//==================================================================================================
//							Beckhoff Automation Poland
//									10.01.2019
//	Wszystkomajacy blok funkcyjny do sterowania osia, 
//	wymagane biblioteki: Tc2_MC2, Tc2_Utilities
// 	v1.0 	|| TC v 3.1.4022.27	 	|| - first edition
//==================================================================================================
{attribute 'reflection'}
FUNCTION_BLOCK FB_McAxisOnlineNC
VAR_IN_OUT
	stMcAxisOnline						: ST_McAxisOnline;
	Axis								: AXIS_REF;
END_VAR
VAR
	mcPower								: MC_Power;
	mcStop								: MC_Stop;
	mcHalt								: MC_Halt;
	mcStopSS1							: MC_Stop;
	mcStopSS2							: MC_Stop;
	mcReset								: MC_Reset;
	mcHome								: MC_Home;
	mcSetPosition						: MC_SetPosition;
	mcJog								: MC_Jog;

	mcMoveAbsolute						: MC_MoveAbsolute;
	mcMoveRelative						: MC_MoveRelative;
	mcMoveVelocity						: MC_MoveVelocity;
	mcMoveModulo						: MC_MoveModulo;
	mcMoveAbsolute2						: MC_MoveAbsolute;
	mcMoveRelative2						: MC_MoveRelative;
	mcMoveVelocity2						: MC_MoveVelocity;
	mcMoveModulo2						: MC_MoveModulo;

	fbNcLimitSwitch						: FB_NcSWLimitSwitchCtrl;
	mcReadParameterSet					: MC_ReadParameterSet;
	// Internal
	bInitialized						: BOOL;
			
	// Initialization
	iInitStep							: INT;
	bInitializationError				: BOOL;
	wInitializationErrorCounter			: WORD;
	bReadParameterSetReady				: BOOL;
	tonDelay							: TON;
	// Re init
	udiOnlineChangeCntOld				: UDINT;
	bOnlineChangeDetected				: BOOL;
	bReInit								: BOOL;
	bReInitialized						: BOOL;
	bReInitializationError				: BOOL;
	{attribute 'instance-path'}
	{attribute 'noinit'}
	sInstancePath						: STRING;
END_VAR

// Device dependent initialization 
ACT_Initialization();
// Device independent commands, mostly NC 
ACT_States();
ACT_SWLimitSwitch();
ACT_Stop();
ACT_Power();
ACT_Homing();
ACT_Jog();
ACT_Move();
ACT_ResetAndDiag();
ACT_SetPosition();
// Device independent error collection
ACT_ErrorCollection();

ACTION ACT_ErrorCollection:
// Error flags
stMcAxisOnline.stError.bDriveError					:= Axis.Status.DriveDeviceError;

stMcAxisOnline.stError.bNcError						:= Axis.Status.Error;

stMcAxisOnline.stError.bFBError						:= stMcAxisOnline.mcPower.bError OR stMcAxisOnline.mcReset.bError OR stMcAxisOnline.mcHome.bError OR stMcAxisOnline.mcJog.bError
													OR stMcAxisOnline.mcHalt.bError OR stMcAxisOnline.mcStop.bError OR stMcAxisOnline.mcSS1.bError OR stMcAxisOnline.mcSS2.bError
													OR stMcAxisOnline.mcMoveAbsolute.bError OR stMcAxisOnline.mcMoveRelative.bError OR stMcAxisOnline.mcMoveVelocity.bError OR stMcAxisOnline.mcMoveModulo.bError
													OR stMcAxisOnline.mcMoveAbsolute2.bError OR stMcAxisOnline.mcMoveRelative2.bError OR stMcAxisOnline.mcMoveVelocity2.bError OR stMcAxisOnline.mcMoveModulo2.bError
													OR stMcAxisOnline.stNcLimitSwitch.bError OR stMcAxisOnline.mcSetPosition.bError;
									
stMcAxisOnline.stError.bCommunicationError			:= stMcAxisOnline.stChannelErrorCode.bError OR stMcAxisOnline.stSetPositionOffset.bError OR stMcAxisOnline.stMotorMonitoring.bError OR stMcAxisOnline.stHoldingBrake.bError;

stMcAxisOnline.stError.bError						:= stMcAxisOnline.stError.bDriveError OR stMcAxisOnline.stError.bNcError OR stMcAxisOnline.stError.bFBError OR stMcAxisOnline.stError.bCommunicationError;
stMcAxisOnline.bError								:= stMcAxisOnline.stError.bError; // Forward one stage up

// Error codes
stMcAxisOnline.stError.uiDriveErrorID 				:= stMcAxisOnline.stChannelErrorCode.uiChannelErrorCode;
stMcAxisOnline.stError.uiDriveErrorIDHex 			:= stMcAxisOnline.stChannelErrorCode.uiChannelErrorCodeHex;

stMcAxisOnline.stError.udiNcErrorID 				:= Axis.Status.ErrorID;
stMcAxisOnline.stError.udiNcErrorIDHex 				:= Axis.Status.ErrorID;
	

stMcAxisOnline.stError.udiFBErrorID 				:= 	stMcAxisOnline.mcPower.udiErrorID + 
														stMcAxisOnline.mcReset.udiErrorID + 
														stMcAxisOnline.mcHome.udiErrorID + 
														stMcAxisOnline.mcJog.udiErrorID +
														stMcAxisOnline.mcHalt.udiErrorID + 
														stMcAxisOnline.mcStop.udiErrorID + 
														stMcAxisOnline.mcSS1.udiErrorID + 
														stMcAxisOnline.mcSS2.udiErrorID +
														stMcAxisOnline.mcMoveAbsolute.udiErrorID + 
														stMcAxisOnline.mcMoveRelative.udiErrorID + 
														stMcAxisOnline.mcMoveVelocity.udiErrorID + 
														stMcAxisOnline.mcMoveModulo.udiErrorID +
														stMcAxisOnline.mcMoveAbsolute2.udiErrorID + 
														stMcAxisOnline.mcMoveRelative2.udiErrorID + 
														stMcAxisOnline.mcMoveVelocity2.udiErrorID + 
														stMcAxisOnline.mcMoveModulo2.udiErrorID +
														stMcAxisOnline.stNcLimitSwitch.udiErrorID + 
														stMcAxisOnline.mcSetPosition.udiErrorID;

stMcAxisOnline.stError.udiFBErrorIDHex 				:= stMcAxisOnline.stError.udiFBErrorID;

stMcAxisOnline.stError.udiErrorID					:= stMcAxisOnline.stSetPositionOffset.udiErrorID;
stMcAxisOnline.stError.uiAdsErrorID					:= stMcAxisOnline.stChannelErrorCode.uiAdsErrId + stMcAxisOnline.stMotorMonitoring.uiAdsErrId + stMcAxisOnline.stHoldingBrake.uiAdsErrId;
stMcAxisOnline.stError.uiSecErrorID					:= stMcAxisOnline.stChannelErrorCode.uiSecErrId + stMcAxisOnline.stMotorMonitoring.uiSecErrId + stMcAxisOnline.stHoldingBrake.uiSecErrId;

stMcAxisOnline.stError.sNcError						:= F_AxErrMsg(stMcAxisOnline.stError.udiNcErrorID);
stMcAxisOnline.stError.sDriveError					:= F_AX5xErrMsg(stMcAxisOnline.stError.uiDriveErrorID);
END_ACTION

ACTION ACT_Homing:
mcHome(		Axis						:= Axis,
			Execute						:= stMcAxisOnline.mcHome.bExecute,
			Position					:= stMcAxisOnline.mcHome.lrPosition,
			HomingMode					:= stMcAxisOnline.mcHome.eHomingMode,
			BufferMode					:= stMcAxisOnline.mcHome.eBufferMode,
			Options						:= stMcAxisOnline.mcHome.stOptions,
			bCalibrationCam				:= stMcAxisOnline.mcHome.bCalibrationCam,
			Done						=> stMcAxisOnline.mcHome.bDone,
			Busy						=> stMcAxisOnline.mcHome.bBusy,
			Active						=> stMcAxisOnline.mcHome.bActive,
			CommandAborted				=> stMcAxisOnline.mcHome.bCommandAborted,
			Error						=> stMcAxisOnline.mcHome.bError,
			ErrorID						=> stMcAxisOnline.mcHome.udiErrorID);
END_ACTION

ACTION ACT_Initialization:
// bInitialized flag is set just once. 
// bReInitialized ise set each time we do online change or request reinit operation
// bDriveAddressReady, bReadParameterSetReady, bDriveRefReady - set just once after successed read

// Online change detection
bOnlineChangeDetected					:= udiOnlineChangeCntOld <> _AppInfo.OnlineChangeCnt;
udiOnlineChangeCntOld 					:= _AppInfo.OnlineChangeCnt;
// Reset init
IF bReInit OR bOnlineChangeDetected THEN
	iInitStep							:= 0;
END_IF

//Initialization process
CASE iInitStep OF
	0:	// Read Parameter Set
		
		stMcAxisOnline.mcReadParameterSet.bExecute		:=	 TRUE;
		iInitStep						:= iInitStep + 10;
		
	10: // Wait for data
	
		IF NOT stMcAxisOnline.mcReadParameterSet.bBusy THEN
			stMcAxisOnline.mcReadParameterSet.bExecute	:=	 FALSE;
			IF stMcAxisOnline.mcReadParameterSet.bDone THEN
				iInitStep 				:= iInitStep + 10;
				bReadParameterSetReady 	:= TRUE;
			ELSE
				iInitStep 				:= 1000;		// Error step
			END_IF
		END_IF	
	
	20: // Success - initialized flag, clear error
		bReInitialized					:= bInitialized;	// TRUE only when it's not first initialization e.g. online change
		bInitialized 					:= TRUE;
		bReInitializationError			:= FALSE;			// TRUE only when it's not first initialization e.g. online change
		bInitializationError			:= FALSE;
		iInitStep 						:= iInitStep + 10;
		
	30: // Idle
	
		;
		
	1000: // Error step
		wInitializationErrorCounter 	:= wInitializationErrorCounter + 1;
		IF wInitializationErrorCounter < 100 THEN
			iInitStep					:= iInitStep + 5;			// Go to delay
		ELSE
			bReInitializationError		:= bInitializationError;	// TRUE only when it's not first initialization e.g. online change
			bInitializationError		:= TRUE;
			bReInitialized				:= FALSE;
			iInitStep 					:= iInitStep + 10;
		END_IF

	1005: // Delay step
		tonDelay(IN:= TRUE, PT:= T#1S);
		IF tonDelay.Q THEN
			tonDelay(IN:= FALSE, PT:= T#1S);
			iInitStep					:= 0;
		END_IF
		
	1010: // Idle after error
		;
	
END_CASE
				
mcReadParameterSet(	Parameter			:= stMcAxisOnline.stAxisParameter,
					Axis				:= Axis,
					Execute				:= stMcAxisOnline.mcReadParameterSet.bExecute,
					Done				=> stMcAxisOnline.mcReadParameterSet.bDone,
					Busy				=> stMcAxisOnline.mcReadParameterSet.bBusy,
					Error				=> stMcAxisOnline.mcReadParameterSet.bError,
					ErrorID				=> stMcAxisOnline.mcReadParameterSet.udiErrorID);
END_ACTION

ACTION ACT_Jog:
// Direct access from bSlow or bFast, if none then free choice
IF stMcAxisOnline.mcJog.bSlowForward OR stMcAxisOnline.mcJog.bSlowBackward THEN
	stMcAxisOnline.mcJog.eMode			:= MC_JOGMODE_STANDARD_SLOW;
ELSIF stMcAxisOnline.mcJog.bFastForward OR stMcAxisOnline.mcJog.bFastBackward THEN
	stMcAxisOnline.mcJog.eMode			:= MC_JOGMODE_STANDARD_FAST;
END_IF

mcJog(		Axis						:= Axis,
			JogForward					:= stMcAxisOnline.mcJog.bJogForward OR stMcAxisOnline.mcJog.bSlowForward OR stMcAxisOnline.mcJog.bFastForward,
			JogBackwards				:= stMcAxisOnline.mcJog.bJogBackwards OR stMcAxisOnline.mcJog.bSlowBackward OR stMcAxisOnline.mcJog.bFastBackward,
			Mode						:= stMcAxisOnline.mcJog.eMode,
			Position					:= stMcAxisOnline.mcJog.lrPosition,
			Velocity					:= stMcAxisOnline.mcJog.lrVelocity,
			Acceleration				:= stMcAxisOnline.mcJog.lrAcceleration,
			Deceleration				:= stMcAxisOnline.mcJog.lrDeceleration,
			Jerk						:= stMcAxisOnline.mcJog.lrJerk,
			Done						=> stMcAxisOnline.mcJog.bDone,
			Busy						=> stMcAxisOnline.mcJog.bBusy,
			Active						=> stMcAxisOnline.mcJog.bActive,
			CommandAborted				=> stMcAxisOnline.mcJog.bCommandAborted,
			Error						=> stMcAxisOnline.mcJog.bError,
			ErrorID						=> stMcAxisOnline.mcJog.udiErrorID);
END_ACTION

ACTION ACT_Move:
{region "Primary"}
mcMoveAbsolute(	Axis					:= Axis,
				Execute					:= stMcAxisOnline.mcMoveAbsolute.bExecute,
				Position				:= stMcAxisOnline.mcMoveAbsolute.lrPosition,
				Velocity				:= stMcAxisOnline.mcMoveAbsolute.lrVelocity,
				Acceleration			:= stMcAxisOnline.mcMoveAbsolute.lrAcceleration,
				Deceleration			:= stMcAxisOnline.mcMoveAbsolute.lrDeceleration,
				Jerk					:= stMcAxisOnline.mcMoveAbsolute.lrJerk,
				BufferMode				:= stMcAxisOnline.mcMoveAbsolute.eBufferMode,
				Options					:= stMcAxisOnline.mcMoveAbsolute.stOptions,
				Done					=> stMcAxisOnline.mcMoveAbsolute.bDone,
				Busy					=> stMcAxisOnline.mcMoveAbsolute.bBusy,
				Active					=> stMcAxisOnline.mcMoveAbsolute.bActive,
				CommandAborted			=> stMcAxisOnline.mcMoveAbsolute.bCommandAborted,
				Error					=> stMcAxisOnline.mcMoveAbsolute.bError,
				ErrorID					=> stMcAxisOnline.mcMoveAbsolute.udiErrorID);

mcMoveRelative(	Axis					:= Axis,
				Execute					:= stMcAxisOnline.mcMoveRelative.bExecute,
				Distance				:= stMcAxisOnline.mcMoveRelative.lrDistance,
				Velocity				:= stMcAxisOnline.mcMoveRelative.lrVelocity,
				Acceleration			:= stMcAxisOnline.mcMoveRelative.lrAcceleration,
				Deceleration			:= stMcAxisOnline.mcMoveRelative.lrDeceleration,
				Jerk					:= stMcAxisOnline.mcMoveRelative.lrJerk,
				BufferMode				:= stMcAxisOnline.mcMoveRelative.eBufferMode,
				Options					:= stMcAxisOnline.mcMoveRelative.stOptions,
				Done					=> stMcAxisOnline.mcMoveRelative.bDone,
				Busy					=> stMcAxisOnline.mcMoveRelative.bBusy,
				Active					=> stMcAxisOnline.mcMoveRelative.bActive,
				CommandAborted			=> stMcAxisOnline.mcMoveRelative.bCommandAborted,
				Error					=> stMcAxisOnline.mcMoveRelative.bError,
				ErrorID					=> stMcAxisOnline.mcMoveRelative.udiErrorID);
				
mcMoveVelocity(	Axis					:= Axis,
				Execute					:= stMcAxisOnline.mcMoveVelocity.bExecute,
				Velocity				:= stMcAxisOnline.mcMoveVelocity.lrVelocity,
				Acceleration			:= stMcAxisOnline.mcMoveVelocity.lrAcceleration,
				Deceleration			:= stMcAxisOnline.mcMoveVelocity.lrDeceleration,
				Jerk					:= stMcAxisOnline.mcMoveVelocity.lrJerk,
				Direction				:= stMcAxisOnline.mcMoveVelocity.eDirection,
				BufferMode				:= stMcAxisOnline.mcMoveVelocity.eBufferMode,
				Options					:= stMcAxisOnline.mcMoveVelocity.stOptions,
				InVelocity				=> stMcAxisOnline.mcMoveVelocity.bInVelocity,
				Busy					=> stMcAxisOnline.mcMoveVelocity.bBusy,
				Active					=> stMcAxisOnline.mcMoveVelocity.bActive,
				CommandAborted			=> stMcAxisOnline.mcMoveVelocity.bCommandAborted,
				Error					=> stMcAxisOnline.mcMoveVelocity.bError,
				ErrorID					=> stMcAxisOnline.mcMoveVelocity.udiErrorID);
stMcAxisOnline.mcMoveVelocity.bDone		:= stMcAxisOnline.mcMoveVelocity.bInVelocity;

mcMoveModulo(	Axis					:= Axis,
				Execute					:= stMcAxisOnline.mcMoveModulo.bExecute,
				Position				:= stMcAxisOnline.mcMoveModulo.lrPosition,
				Velocity				:= stMcAxisOnline.mcMoveModulo.lrVelocity,
				Acceleration			:= stMcAxisOnline.mcMoveModulo.lrAcceleration,
				Deceleration			:= stMcAxisOnline.mcMoveModulo.lrDeceleration,
				Jerk					:= stMcAxisOnline.mcMoveModulo.lrJerk,
				Direction				:= stMcAxisOnline.mcMoveModulo.eDirection,
				BufferMode				:= stMcAxisOnline.mcMoveModulo.eBufferMode,
				Options					:= stMcAxisOnline.mcMoveModulo.stOptions,
				Done					=> stMcAxisOnline.mcMoveModulo.bDone,
				Busy					=> stMcAxisOnline.mcMoveModulo.bBusy,
				Active					=> stMcAxisOnline.mcMoveModulo.bActive,
				CommandAborted			=> stMcAxisOnline.mcMoveModulo.bCommandAborted,
				Error					=> stMcAxisOnline.mcMoveModulo.bError,
				ErrorID					=> stMcAxisOnline.mcMoveModulo.udiErrorID);
{endregion}
{region "Secondary"}
mcMoveAbsolute2(Axis					:= Axis,
				Execute					:= stMcAxisOnline.mcMoveAbsolute2.bExecute,
				Position				:= stMcAxisOnline.mcMoveAbsolute2.lrPosition,
				Velocity				:= stMcAxisOnline.mcMoveAbsolute2.lrVelocity,
				Acceleration			:= stMcAxisOnline.mcMoveAbsolute2.lrAcceleration,
				Deceleration			:= stMcAxisOnline.mcMoveAbsolute2.lrDeceleration,
				Jerk					:= stMcAxisOnline.mcMoveAbsolute2.lrJerk,
				BufferMode				:= stMcAxisOnline.mcMoveAbsolute2.eBufferMode,
				Options					:= stMcAxisOnline.mcMoveAbsolute2.stOptions,
				Done					=> stMcAxisOnline.mcMoveAbsolute2.bDone,
				Busy					=> stMcAxisOnline.mcMoveAbsolute2.bBusy,
				Active					=> stMcAxisOnline.mcMoveAbsolute2.bActive,
				CommandAborted			=> stMcAxisOnline.mcMoveAbsolute2.bCommandAborted,
				Error					=> stMcAxisOnline.mcMoveAbsolute2.bError,
				ErrorID					=> stMcAxisOnline.mcMoveAbsolute2.udiErrorID);

mcMoveRelative2(Axis					:= Axis,
				Execute					:= stMcAxisOnline.mcMoveRelative2.bExecute,
				Distance				:= stMcAxisOnline.mcMoveRelative2.lrDistance,
				Velocity				:= stMcAxisOnline.mcMoveRelative2.lrVelocity,
				Acceleration			:= stMcAxisOnline.mcMoveRelative2.lrAcceleration,
				Deceleration			:= stMcAxisOnline.mcMoveRelative2.lrDeceleration,
				Jerk					:= stMcAxisOnline.mcMoveRelative2.lrJerk,
				BufferMode				:= stMcAxisOnline.mcMoveRelative2.eBufferMode,
				Options					:= stMcAxisOnline.mcMoveRelative2.stOptions,
				Done					=> stMcAxisOnline.mcMoveRelative2.bDone,
				Busy					=> stMcAxisOnline.mcMoveRelative2.bBusy,
				Active					=> stMcAxisOnline.mcMoveRelative2.bActive,
				CommandAborted			=> stMcAxisOnline.mcMoveRelative2.bCommandAborted,
				Error					=> stMcAxisOnline.mcMoveRelative2.bError,
				ErrorID					=> stMcAxisOnline.mcMoveRelative2.udiErrorID);
				
mcMoveVelocity2(Axis					:= Axis,
				Execute					:= stMcAxisOnline.mcMoveVelocity2.bExecute,
				Velocity				:= stMcAxisOnline.mcMoveVelocity2.lrVelocity,
				Acceleration			:= stMcAxisOnline.mcMoveVelocity2.lrAcceleration,
				Deceleration			:= stMcAxisOnline.mcMoveVelocity2.lrDeceleration,
				Jerk					:= stMcAxisOnline.mcMoveVelocity2.lrJerk,
				Direction				:= stMcAxisOnline.mcMoveVelocity2.eDirection,
				BufferMode				:= stMcAxisOnline.mcMoveVelocity2.eBufferMode,
				Options					:= stMcAxisOnline.mcMoveVelocity2.stOptions,
				InVelocity				=> stMcAxisOnline.mcMoveVelocity2.bInVelocity,
				Busy					=> stMcAxisOnline.mcMoveVelocity2.bBusy,
				Active					=> stMcAxisOnline.mcMoveVelocity2.bActive,
				CommandAborted			=> stMcAxisOnline.mcMoveVelocity2.bCommandAborted,
				Error					=> stMcAxisOnline.mcMoveVelocity2.bError,
				ErrorID					=> stMcAxisOnline.mcMoveVelocity2.udiErrorID);
stMcAxisOnline.mcMoveVelocity2.bDone	:= stMcAxisOnline.mcMoveVelocity2.bInVelocity;

mcMoveModulo2(	Axis					:= Axis,
				Execute					:= stMcAxisOnline.mcMoveModulo2.bExecute,
				Position				:= stMcAxisOnline.mcMoveModulo2.lrPosition,
				Velocity				:= stMcAxisOnline.mcMoveModulo2.lrVelocity,
				Acceleration			:= stMcAxisOnline.mcMoveModulo2.lrAcceleration,
				Deceleration			:= stMcAxisOnline.mcMoveModulo2.lrDeceleration,
				Jerk					:= stMcAxisOnline.mcMoveModulo2.lrJerk,
				Direction				:= stMcAxisOnline.mcMoveModulo2.eDirection,
				BufferMode				:= stMcAxisOnline.mcMoveModulo2.eBufferMode,
				Options					:= stMcAxisOnline.mcMoveModulo2.stOptions,
				Done					=> stMcAxisOnline.mcMoveModulo2.bDone,
				Busy					=> stMcAxisOnline.mcMoveModulo2.bBusy,
				Active					=> stMcAxisOnline.mcMoveModulo2.bActive,
				CommandAborted			=> stMcAxisOnline.mcMoveModulo2.bCommandAborted,
				Error					=> stMcAxisOnline.mcMoveModulo2.bError,
				ErrorID					=> stMcAxisOnline.mcMoveModulo2.udiErrorID);
{endregion}
END_ACTION

ACTION ACT_Power:
mcPower(	Axis						:= Axis,									//
			Enable						:= stMcAxisOnline.mcPower.bEnable,
			Enable_Positive				:= stMcAxisOnline.mcPower.bEnable_Positive,
			Enable_Negative				:= stMcAxisOnline.mcPower.bEnable_Negative,
			Override					:= stMcAxisOnline.mcPower.lrOverride,
			BufferMode					:= stMcAxisOnline.mcPower.eBufferMode,
			Options						:= stMcAxisOnline.mcPower.stOptions,
			Status						=> stMcAxisOnline.mcPower.bStatus,
			Busy						=> stMcAxisOnline.mcPower.bBusy,
			Active						=> stMcAxisOnline.mcPower.bActive,
			Error						=> stMcAxisOnline.mcPower.bError,
			ErrorID						=> stMcAxisOnline.mcPower.udiErrorID);
END_ACTION

ACTION ACT_ResetAndDiag:
mcReset(
	Axis						:= Axis,
	Execute						:= stMcAxisOnline.mcReset.bExecute,
	Done						=> stMcAxisOnline.mcReset.bDone,
	Busy						=> stMcAxisOnline.mcReset.bBusy,
	Error						=> stMcAxisOnline.mcReset.bError,
	ErrorID						=> stMcAxisOnline.mcReset.udiErrorID);
END_ACTION

ACTION ACT_SetPosition:
mcSetPosition(		Axis				:= Axis,
					Execute				:= stMcAxisOnline.mcSetPosition.bExecute,
					Position			:= stMcAxisOnline.mcSetPosition.lrPosition,
					Mode				:= stMcAxisOnline.mcSetPosition.bMode,
					Options				:= stMcAxisOnline.mcSetPosition.stOptions,
					Done				=> stMcAxisOnline.mcSetPosition.bDone,
					Busy				=> stMcAxisOnline.mcSetPosition.bBusy,
					Error				=> stMcAxisOnline.mcSetPosition.bError,
					ErrorID				=> stMcAxisOnline.mcSetPosition.udiErrorID);
END_ACTION

ACTION ACT_States:
// Read States and forward main states
Axis.ReadStatus();
stMcAxisOnline.stStatus.stAxisStatus		:= Axis.Status;
stMcAxisOnline.stStatus.dwAxisId			:= Axis.NcToPlc.AxisId;
stMcAxisOnline.stStatus.bNcError			:= Axis.Status.Error;
stMcAxisOnline.stStatus.udiNcErrorCode		:= Axis.Status.ErrorID;
stMcAxisOnline.stStatus.udiNcErrorCodeHex	:= Axis.Status.ErrorID;

stMcAxisOnline.stStatus.sAxisName			:= stMcAxisOnline.stAxisParameter.sAxisName;
stMcAxisOnline.stStatus.lrActPos			:= Axis.NcToPlc.ActPos;
stMcAxisOnline.stStatus.lrModuloActPos		:= Axis.NcToPlc.ModuloActPos;
stMcAxisOnline.stStatus.lrActVelo			:= Axis.NcToPlc.ActVelo;
stMcAxisOnline.stStatus.lrActAcc			:= Axis.NcToPlc.ActAcc;
stMcAxisOnline.stStatus.lrActTorque			:= Axis.NcToPlc.ActTorque;
stMcAxisOnline.stStatus.lrPosDiff			:= Axis.NcToPlc.PosDiff;
stMcAxisOnline.stStatus.lrSetPos			:= Axis.NcToPlc.SetPos;
stMcAxisOnline.stStatus.lrSetVelo			:= Axis.NcToPlc.SetVelo;
stMcAxisOnline.stStatus.lrSetAcc			:= Axis.NcToPlc.SetAcc;
stMcAxisOnline.stStatus.lrSetTorque			:= Axis.NcToPlc.SetTorque;
stMcAxisOnline.stStatus.lrPosDiff			:= Axis.NcToPlc.PosDiff;
stMcAxisOnline.stStatus.bAxisReady			:= Axis.Status.Operational;
stMcAxisOnline.stStatus.bHomed				:= Axis.Status.Homed;
stMcAxisOnline.stStatus.bCoupled			:= Axis.Status.Coupled;

// zezwolenie na zjazd z krancowki hw
Axis.PlcToNc.ControlDWord.8				:= stMcAxisOnline.stStatus.bAcceptBlockedDrive;
END_ACTION

ACTION ACT_Stop:
mcHalt(		Axis						:= Axis,
			Execute						:= stMcAxisOnline.mcHalt.bExecute,
			Deceleration				:= stMcAxisOnline.mcHalt.lrDeceleration,
			Jerk						:= stMcAxisOnline.mcHalt.lrJerk,
			BufferMode					:= stMcAxisOnline.mcHalt.eBufferMode,
			Options						:= stMcAxisOnline.mcHalt.stOptions,
			Done						=> stMcAxisOnline.mcHalt.bDone,
			Busy						=> stMcAxisOnline.mcHalt.bBusy,
			Active						=> stMcAxisOnline.mcHalt.bActive,
			CommandAborted				=> stMcAxisOnline.mcHalt.bCommandAborted,
			Error						=> stMcAxisOnline.mcHalt.bError,
			ErrorID						=> stMcAxisOnline.mcHalt.udiErrorID);
			
mcStop(		Axis						:= Axis,
			Execute						:= stMcAxisOnline.mcStop.bExecute,
			Deceleration				:= stMcAxisOnline.mcStop.lrDeceleration,
			Jerk						:= stMcAxisOnline.mcStop.lrJerk,
			Options						:= stMcAxisOnline.mcStop.stOptions,
			Done						=> stMcAxisOnline.mcStop.bDone,
			Busy						=> stMcAxisOnline.mcStop.bBusy,
			Active						=> stMcAxisOnline.mcStop.bActive,
			CommandAborted				=> stMcAxisOnline.mcStop.bCommandAborted,
			Error						=> stMcAxisOnline.mcStop.bError,
			ErrorID						=> stMcAxisOnline.mcStop.udiErrorID);
			
mcStopSS2(	Axis						:= Axis,
			Execute						:= stMcAxisOnline.mcSS2.bExecute,
			Deceleration				:= stMcAxisOnline.mcSS2.lrDeceleration,
			Jerk						:= stMcAxisOnline.mcSS2.lrJerk,
			Options						:= stMcAxisOnline.mcSS2.stOptions,
			Done						=> stMcAxisOnline.mcSS2.bDone,
			Busy						=> stMcAxisOnline.mcSS2.bBusy,
			Active						=> stMcAxisOnline.mcSS2.bActive,
			CommandAborted				=> stMcAxisOnline.mcSS2.bCommandAborted,
			Error						=> stMcAxisOnline.mcSS2.bError,
			ErrorID						=> stMcAxisOnline.mcSS2.udiErrorID);
			
mcStopSS1(	Axis						:= Axis,
			Execute						:= stMcAxisOnline.mcSS1.bExecute,
			Deceleration				:= stMcAxisOnline.mcSS1.lrDeceleration,
			Jerk						:= stMcAxisOnline.mcSS1.lrJerk,
			Options						:= stMcAxisOnline.mcSS1.stOptions,
			Done						=> stMcAxisOnline.mcSS1.bDone,
			Busy						=> stMcAxisOnline.mcSS1.bBusy,
			Active						=> stMcAxisOnline.mcSS1.bActive,
			CommandAborted				=> stMcAxisOnline.mcSS1.bCommandAborted,
			Error						=> stMcAxisOnline.mcSS1.bError,
			ErrorID						=> stMcAxisOnline.mcSS1.udiErrorID);
// SS1 - after MC_Stop function we have to disable drive			
stMcAxisOnline.mcPower.bEnable R= stMcAxisOnline.mcPower.bEnable_Positive R= stMcAxisOnline.mcPower.bEnable_Negative R= (stMcAxisOnline.mcSS1.bDone OR stMcAxisOnline.mcSS1.bCommandAborted OR stMcAxisOnline.mcSS1.bError);
END_ACTION

ACTION ACT_SWLimitSwitch:
fbNcLimitSwitch(	udiAxisID		:= Axis.NcToPlc.AxisId, 
					bRead			:= stMcAxisOnline.stNcLimitSwitch.bRead, 
					bWrite			:= stMcAxisOnline.stNcLimitSwitch.bWrite, 
					bReset			:= stMcAxisOnline.stNcLimitSwitch.bReset, 
					lrSetMinPos		:= stMcAxisOnline.stNcLimitSwitch.lrSetMinPos, 
					lrSetMaxPos		:= stMcAxisOnline.stNcLimitSwitch.lrSetMaxPos, 
					bSetMinMon		:= stMcAxisOnline.stNcLimitSwitch.bSetMinMon, 
					bSetMaxMon		:= stMcAxisOnline.stNcLimitSwitch.bSetMaxMon, 
					bBusy			=> stMcAxisOnline.stNcLimitSwitch.bBusy, 
					bError			=> stMcAxisOnline.stNcLimitSwitch.bError, 
					udiErrorID		=> stMcAxisOnline.stNcLimitSwitch.udiErrorID, 
					lrActMinPos		=> stMcAxisOnline.stNcLimitSwitch.lrActMinPos, 
					lrActMaxPos		=> stMcAxisOnline.stNcLimitSwitch.lrActMaxPos, 
					bActMinMon		=> stMcAxisOnline.stNcLimitSwitch.bActMinMon, 
					bActMaxMon		=> stMcAxisOnline.stNcLimitSwitch.bActMaxMon);
END_ACTION

END_FUNCTION_BLOCK

(* stored: Version 1.1.0.1, ProductVersion 3.1.4026.13, FileIdentifier 92071da508248f05061f8d92f02c4291c7995f04, FileSignature 4aedaf75a014b489becb4c6bbaa2dec3ef74b381865ab1dbc42d88dbe71818d855562e4b94a9dee37d6ad46c712f9dbdb582db1370f36a52336cb476b604594b86de955be351fb5914f52ff121661c1aa53d11df68984254ec3883d99ddd731059b535fefd6f329dee3e8a63076680d0597f245628c79d8b6eeb9931fb498a56d434e373c414ff15873039c4e2509a37d59a018ce371874c8600082b22cf03b6af18ecaa05743ef5b5218520de3f62d68d6bc71ffbc619057bbce154762cec00df5e339634c70d08e69fbcea7c1dfaf00a022973f5cfb4ca3900e587a4d79935d7c50a4fa88b60629b489672614e0546eebd07143ab1335422f07e6f1134628d
   POU FB_McAxisOnlineNC: Id {b4626b7f-b730-4c5f-9617-35502c9fa0f9}, SpecialFunc None
   Action ACT_ErrorCollection: Id {93a18eec-e7c3-45ab-ba23-46ad6b21ec58}
   Action ACT_Homing: Id {302d006c-ac02-4c87-bf93-bba1abe49fd7}
   Action ACT_Initialization: Id {e47a96a3-e267-44ea-999c-9d52f7d5d3d9}
   Action ACT_Jog: Id {7a99a723-8c90-4b7c-813f-f0e263f9538a}
   Action ACT_Move: Id {d853b265-1265-4c4a-a2a7-5e33120acf4b}
   Action ACT_Power: Id {39eaba19-b29b-4915-83fd-52a5d2e72160}
   Action ACT_ResetAndDiag: Id {06eeddfa-336c-41e7-8159-b1e91414fac1}
   Action ACT_SetPosition: Id {9e842a73-58b5-4efd-ac79-b2d610940eb2}
   Action ACT_States: Id {e72c0910-9a7d-44ad-97fa-1103c6d79ea8}
   Action ACT_Stop: Id {0fe838ab-18f6-4e70-a174-0b0283acd990}
   Action ACT_SWLimitSwitch: Id {24d5ed38-2863-45bb-894f-f4eccbf166ef} *)
